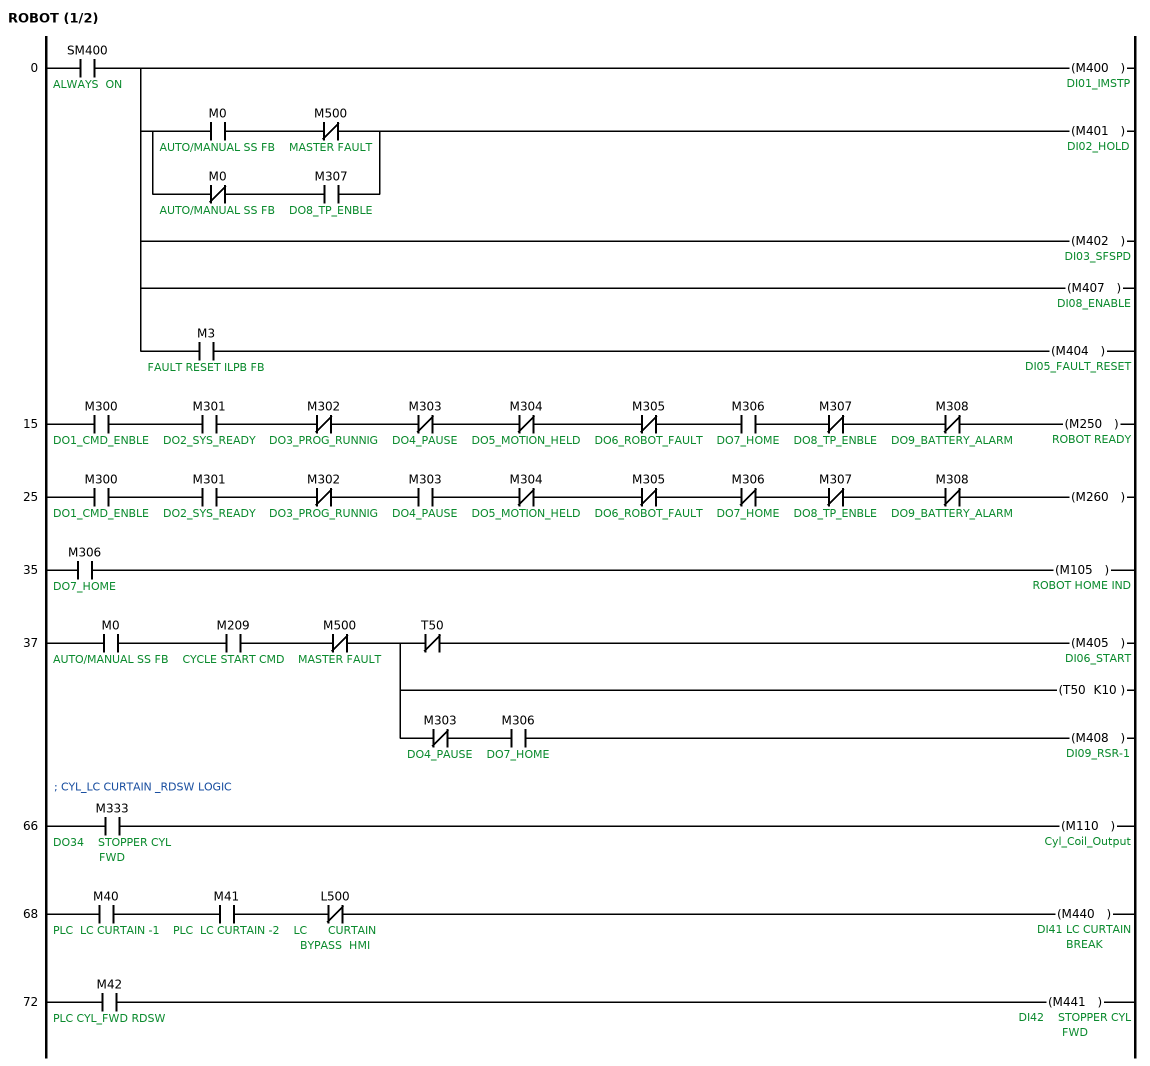
0     LD      SM400  ; ALWAYS  ON
      OUT     M400  ; DI01_IMSTP
      MPS
      LD      M0  ; AUTO/MANUAL SS FB
      ANI     M500  ; MASTER FAULT
      LDI     M0  ; AUTO/MANUAL SS FB
      AND     M307  ; DO8_TP_ENBLE
      ORB
      ANB
      OUT     M401  ; DI02_HOLD
      MPP
      OUT     M402  ; DI03_SFSPD
      OUT     M407  ; DI08_ENABLE
      AND     M3  ; FAULT RESET ILPB FB
      OUT     M404  ; DI05_FAULT_RESET
15    LD      M300  ; DO1_CMD_ENBLE
      AND     M301  ; DO2_SYS_READY
      ANI     M302  ; DO3_PROG_RUNNIG
      ANI     M303  ; DO4_PAUSE
      ANI     M304  ; DO5_MOTION_HELD
      ANI     M305  ; DO6_ROBOT_FAULT
      AND     M306  ; DO7_HOME
      ANI     M307  ; DO8_TP_ENBLE
      ANI     M308  ; DO9_BATTERY_ALARM
      OUT     M250  ; ROBOT READY
25    LD      M300  ; DO1_CMD_ENBLE
      AND     M301  ; DO2_SYS_READY
      ANI     M302  ; DO3_PROG_RUNNIG
      AND     M303  ; DO4_PAUSE
      ANI     M304  ; DO5_MOTION_HELD
      ANI     M305  ; DO6_ROBOT_FAULT
      ANI     M306  ; DO7_HOME
      ANI     M307  ; DO8_TP_ENBLE
      ANI     M308  ; DO9_BATTERY_ALARM
      OUT     M260
35    LD      M306  ; DO7_HOME
      OUT     M105  ; ROBOT HOME IND
37    LD      M0  ; AUTO/MANUAL SS FB
      AND     M209  ; CYCLE START CMD
      ANI     M500  ; MASTER FAULT
      MPS
      ANI     T50
      OUT     M405  ; DI06_START
      MPP
      OUT     T50 K10
      ANI     M303  ; DO4_PAUSE
      AND     M306  ; DO7_HOME
      OUT     M408  ; DI09_RSR-1
; CYL_LC CURTAIN _RDSW LOGIC
66    LD      M333  ; DO34    STOPPER CYL FWD
      OUT     M110  ; Cyl_Coil_Output
68    LD      M40  ; PLC  LC CURTAIN -1
      AND     M41  ; PLC  LC CURTAIN -2
      ANI     L500  ; LC      CURTAIN BYPASS  HMI
      OUT     M440  ; DI41 LC CURTAIN BREAK
72    LD      M42  ; PLC CYL_FWD RDSW
      OUT     M441  ; DI42    STOPPER CYL FWD
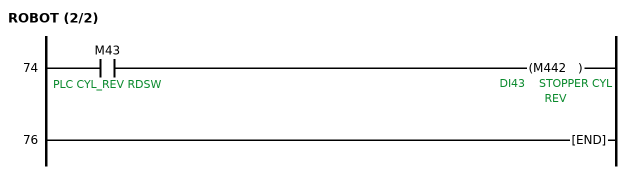
74    LD      M43  ; PLC CYL_REV RDSW
      OUT     M442  ; DI43    STOPPER CYL REV
76    END
END_PROGRAM

PROGRAM CONTROL
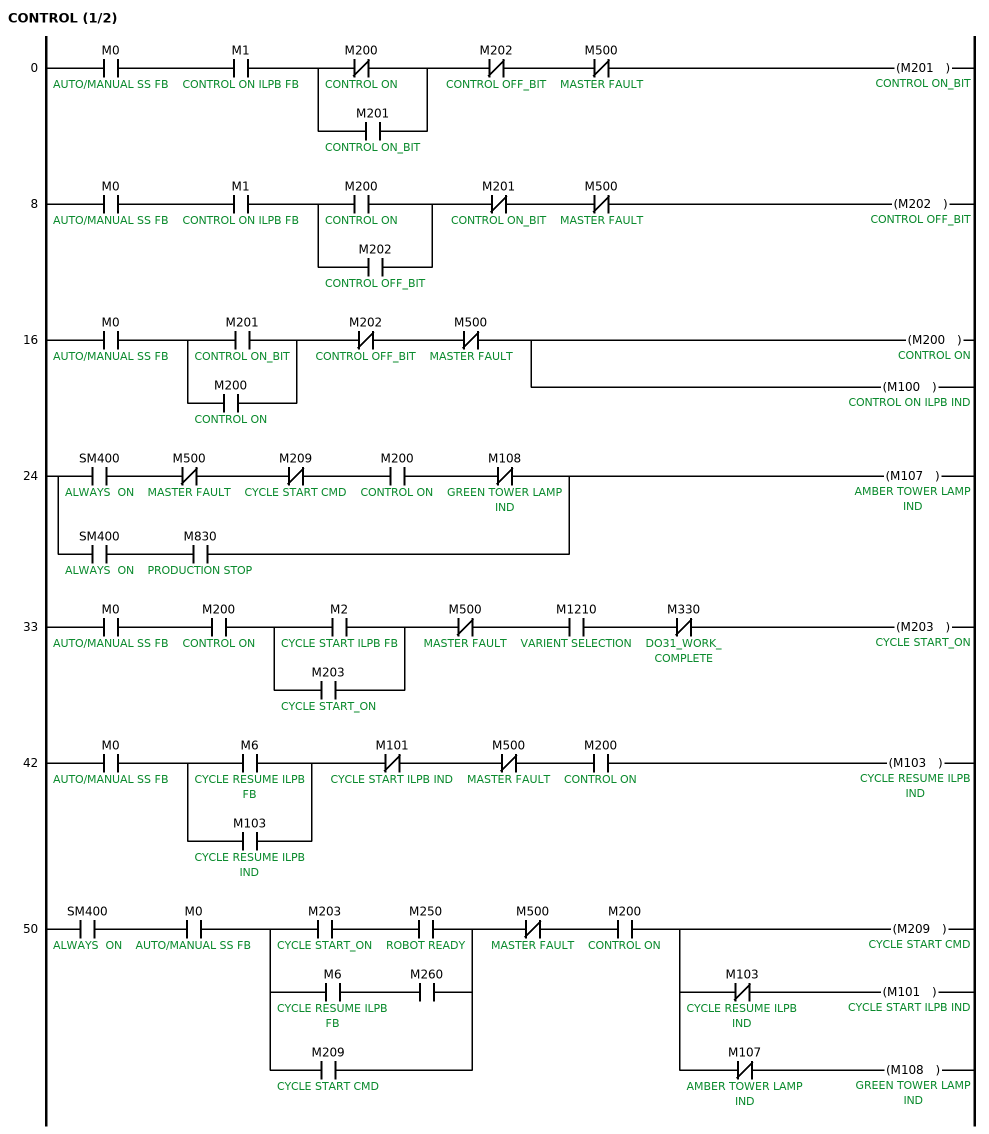
0     LD      M0  ; AUTO/MANUAL SS FB
      AND     M1  ; CONTROL ON ILPB FB
      LDI     M200  ; CONTROL ON
      OR      M201  ; CONTROL ON_BIT
      ANB
      ANI     M202  ; CONTROL OFF_BIT
      ANI     M500  ; MASTER FAULT
      OUT     M201  ; CONTROL ON_BIT
8     LD      M0  ; AUTO/MANUAL SS FB
      AND     M1  ; CONTROL ON ILPB FB
      LD      M200  ; CONTROL ON
      OR      M202  ; CONTROL OFF_BIT
      ANB
      ANI     M201  ; CONTROL ON_BIT
      ANI     M500  ; MASTER FAULT
      OUT     M202  ; CONTROL OFF_BIT
16    LD      M0  ; AUTO/MANUAL SS FB
      LD      M201  ; CONTROL ON_BIT
      OR      M200  ; CONTROL ON
      ANB
      ANI     M202  ; CONTROL OFF_BIT
      ANI     M500  ; MASTER FAULT
      OUT     M200  ; CONTROL ON
      OUT     M100  ; CONTROL ON ILPB IND
24    LD      SM400  ; ALWAYS  ON
      ANI     M500  ; MASTER FAULT
      ANI     M209  ; CYCLE START CMD
      AND     M200  ; CONTROL ON
      ANI     M108  ; GREEN TOWER LAMP IND
      LD      SM400  ; ALWAYS  ON
      AND     M830  ; PRODUCTION STOP
      ORB
      OUT     M107  ; AMBER TOWER LAMP IND
33    LD      M0  ; AUTO/MANUAL SS FB
      AND     M200  ; CONTROL ON
      LD      M2  ; CYCLE START ILPB FB
      OR      M203  ; CYCLE START_ON
      ANB
      ANI     M500  ; MASTER FAULT
      AND     M1210  ; VARIENT SELECTION
      ANI     M330  ; DO31_WORK_COMPLETE
      OUT     M203  ; CYCLE START_ON
42    LD      M0  ; AUTO/MANUAL SS FB
      LD      M6  ; CYCLE RESUME ILPB FB
      OR      M103  ; CYCLE RESUME ILPB IND
      ANB
      ANI     M101  ; CYCLE START ILPB IND
      ANI     M500  ; MASTER FAULT
      AND     M200  ; CONTROL ON
      OUT     M103  ; CYCLE RESUME ILPB IND
50    LD      SM400  ; ALWAYS  ON
      AND     M0  ; AUTO/MANUAL SS FB
      LD      M203  ; CYCLE START_ON
      AND     M250  ; ROBOT READY
      LD      M6  ; CYCLE RESUME ILPB FB
      AND     M260
      ORB
      OR      M209  ; CYCLE START CMD
      ANB
      ANI     M500  ; MASTER FAULT
      AND     M200  ; CONTROL ON
      OUT     M209  ; CYCLE START CMD
      MPS
      ANI     M103  ; CYCLE RESUME ILPB IND
      OUT     M101  ; CYCLE START ILPB IND
      MPP
      ANI     M107  ; AMBER TOWER LAMP IND
      OUT     M108  ; GREEN TOWER LAMP IND
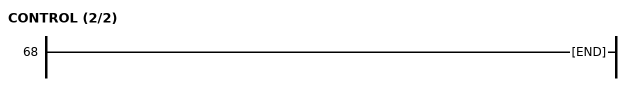
68    END
END_PROGRAM

PROGRAM FAULT
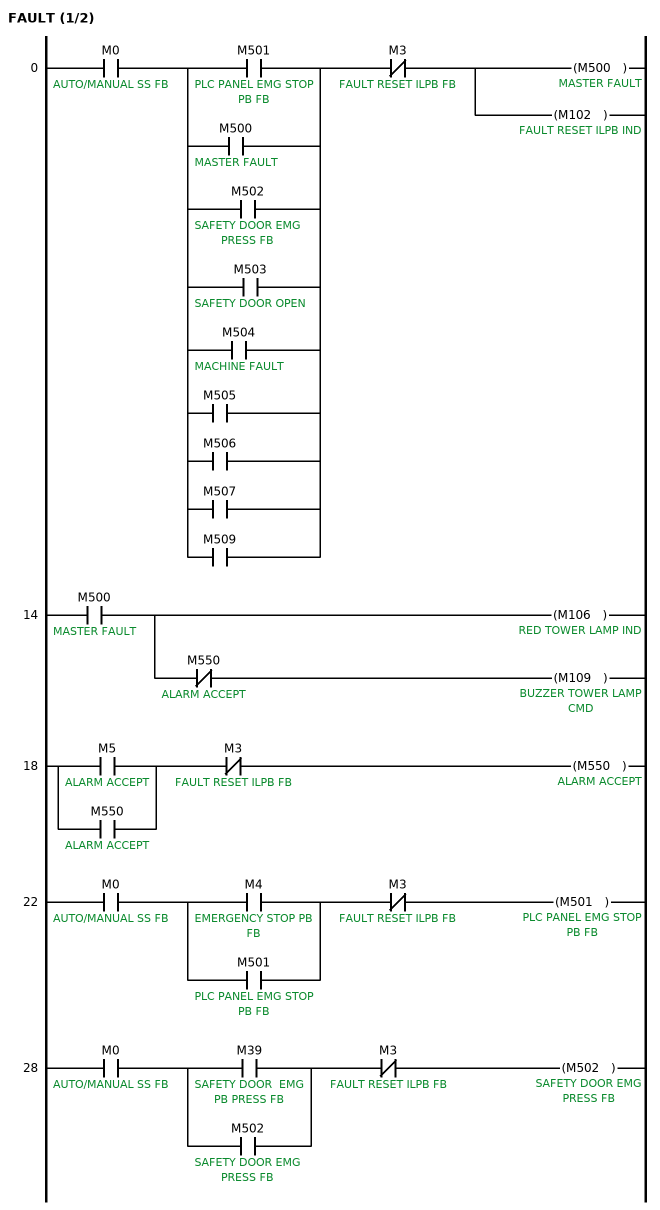
0     LD      M0  ; AUTO/MANUAL SS FB
      LD      M501  ; PLC PANEL EMG STOP PB FB
      OR      M500  ; MASTER FAULT
      OR      M502  ; SAFETY DOOR EMG PRESS FB
      OR      M503  ; SAFETY DOOR OPEN
      OR      M504  ; MACHINE FAULT
      OR      M505
      OR      M506
      OR      M507
      OR      M509
      ANB
      ANI     M3  ; FAULT RESET ILPB FB
      OUT     M500  ; MASTER FAULT
      OUT     M102  ; FAULT RESET ILPB IND
14    LD      M500  ; MASTER FAULT
      OUT     M106  ; RED TOWER LAMP IND
      ANI     M550  ; ALARM ACCEPT
      OUT     M109  ; BUZZER TOWER LAMP CMD
18    LD      M5  ; ALARM ACCEPT
      OR      M550  ; ALARM ACCEPT
      ANI     M3  ; FAULT RESET ILPB FB
      OUT     M550  ; ALARM ACCEPT
22    LD      M0  ; AUTO/MANUAL SS FB
      LD      M4  ; EMERGENCY STOP PB FB
      OR      M501  ; PLC PANEL EMG STOP PB FB
      ANB
      ANI     M3  ; FAULT RESET ILPB FB
      OUT     M501  ; PLC PANEL EMG STOP PB FB
28    LD      M0  ; AUTO/MANUAL SS FB
      LD      M39  ; SAFETY DOOR  EMG PB PRESS FB
      OR      M502  ; SAFETY DOOR EMG PRESS FB
      ANB
      ANI     M3  ; FAULT RESET ILPB FB
      OUT     M502  ; SAFETY DOOR EMG PRESS FB
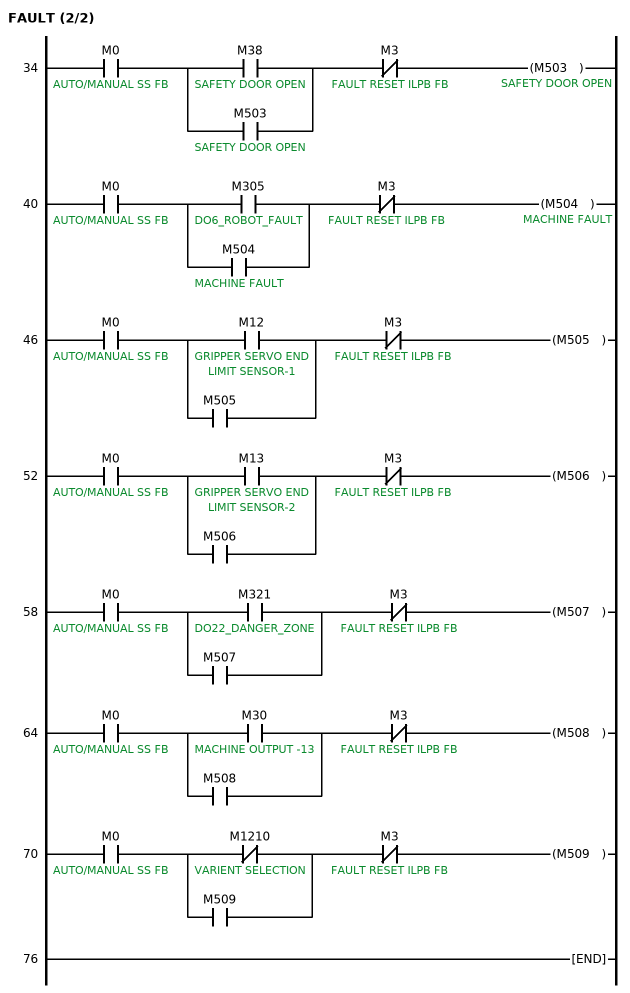
34    LD      M0  ; AUTO/MANUAL SS FB
      LD      M38  ; SAFETY DOOR OPEN
      OR      M503  ; SAFETY DOOR OPEN
      ANB
      ANI     M3  ; FAULT RESET ILPB FB
      OUT     M503  ; SAFETY DOOR OPEN
40    LD      M0  ; AUTO/MANUAL SS FB
      LD      M305  ; DO6_ROBOT_FAULT
      OR      M504  ; MACHINE FAULT
      ANB
      ANI     M3  ; FAULT RESET ILPB FB
      OUT     M504  ; MACHINE FAULT
46    LD      M0  ; AUTO/MANUAL SS FB
      LD      M12  ; GRIPPER SERVO END LIMIT SENSOR-1
      OR      M505
      ANB
      ANI     M3  ; FAULT RESET ILPB FB
      OUT     M505
52    LD      M0  ; AUTO/MANUAL SS FB
      LD      M13  ; GRIPPER SERVO END LIMIT SENSOR-2
      OR      M506
      ANB
      ANI     M3  ; FAULT RESET ILPB FB
      OUT     M506
58    LD      M0  ; AUTO/MANUAL SS FB
      LD      M321  ; DO22_DANGER_ZONE
      OR      M507
      ANB
      ANI     M3  ; FAULT RESET ILPB FB
      OUT     M507
64    LD      M0  ; AUTO/MANUAL SS FB
      LD      M30  ; MACHINE OUTPUT -13
      OR      M508
      ANB
      ANI     M3  ; FAULT RESET ILPB FB
      OUT     M508
70    LD      M0  ; AUTO/MANUAL SS FB
      LDI     M1210  ; VARIENT SELECTION
      OR      M509
      ANB
      ANI     M3  ; FAULT RESET ILPB FB
      OUT     M509
76    END
END_PROGRAM

PROGRAM MACHINE
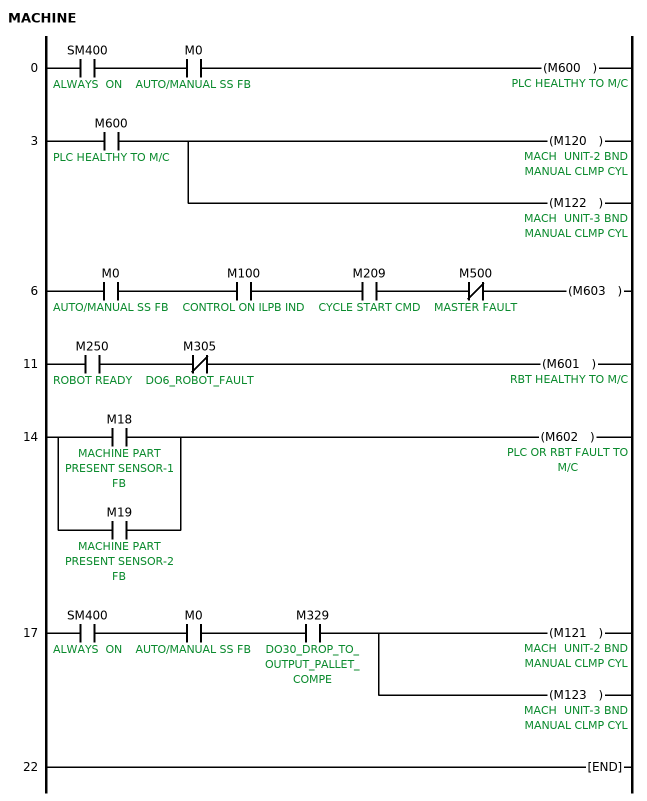
0     LD      SM400  ; ALWAYS  ON
      AND     M0  ; AUTO/MANUAL SS FB
      OUT     M600  ; PLC HEALTHY TO M/C
3     LD      M600  ; PLC HEALTHY TO M/C
      OUT     M120  ; MACH  UNIT-2 BND MANUAL CLMP CYL
      OUT     M122  ; MACH  UNIT-3 BND MANUAL CLMP CYL
6     LD      M0  ; AUTO/MANUAL SS FB
      AND     M100  ; CONTROL ON ILPB IND
      AND     M209  ; CYCLE START CMD
      ANI     M500  ; MASTER FAULT
      OUT     M603
11    LD      M250  ; ROBOT READY
      ANI     M305  ; DO6_ROBOT_FAULT
      OUT     M601  ; RBT HEALTHY TO M/C
14    LD      M18  ; MACHINE PART PRESENT SENSOR-1 FB
      OR      M19  ; MACHINE PART PRESENT SENSOR-2 FB
      OUT     M602  ; PLC OR RBT FAULT TO M/C
17    LD      SM400  ; ALWAYS  ON
      AND     M0  ; AUTO/MANUAL SS FB
      AND     M329  ; DO30_DROP_TO_OUTPUT_PALLET_COMPE
      OUT     M121  ; MACH  UNIT-2 BND MANUAL CLMP CYL
      OUT     M123  ; MACH  UNIT-3 BND MANUAL CLMP CYL
22    END
END_PROGRAM

PROGRAM HMI
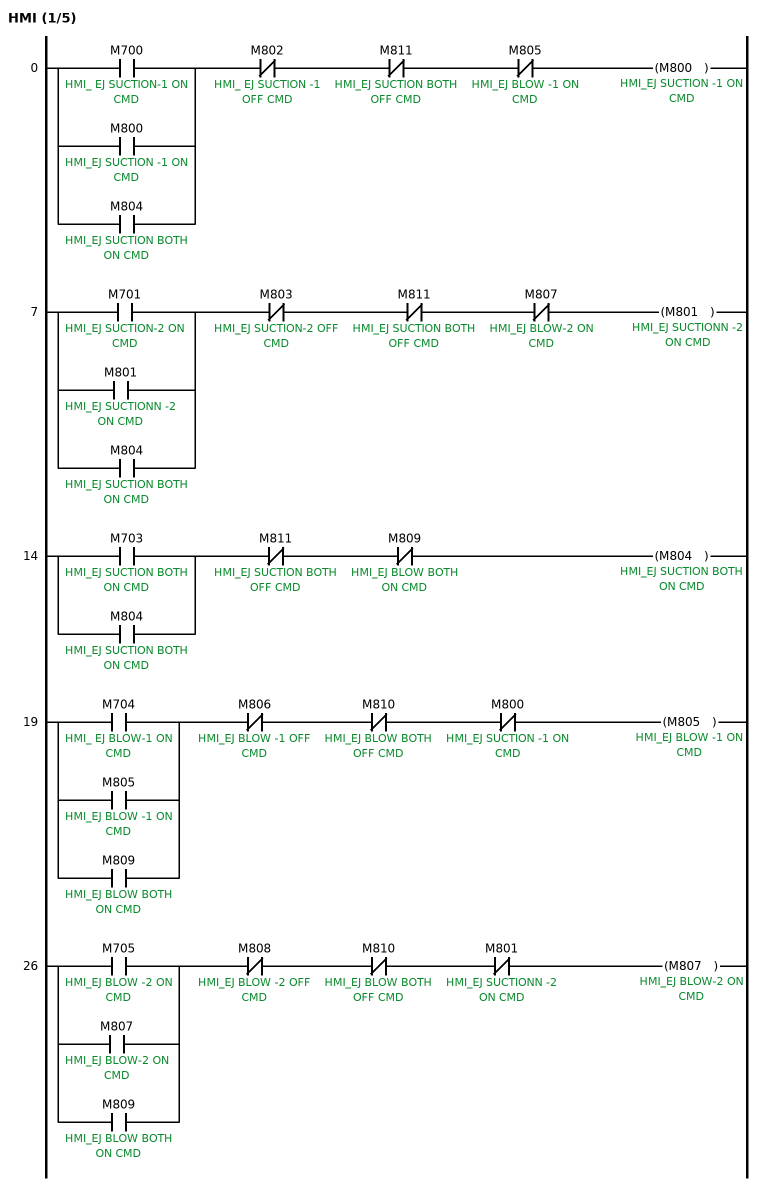
0     LD      M700  ; HMI_ EJ SUCTION-1 ON CMD
      OR      M800  ; HMI_EJ SUCTION -1 ON CMD
      OR      M804  ; HMI_EJ SUCTION BOTH ON CMD
      ANI     M802  ; HMI_ EJ SUCTION -1 OFF CMD
      ANI     M811  ; HMI_EJ SUCTION BOTH OFF CMD
      ANI     M805  ; HMI_EJ BLOW -1 ON CMD
      OUT     M800  ; HMI_EJ SUCTION -1 ON CMD
7     LD      M701  ; HMI_EJ SUCTION-2 ON CMD
      OR      M801  ; HMI_EJ SUCTIONN -2 ON CMD
      OR      M804  ; HMI_EJ SUCTION BOTH ON CMD
      ANI     M803  ; HMI_EJ SUCTION-2 OFF CMD
      ANI     M811  ; HMI_EJ SUCTION BOTH OFF CMD
      ANI     M807  ; HMI_EJ BLOW-2 ON CMD
      OUT     M801  ; HMI_EJ SUCTIONN -2 ON CMD
14    LD      M703  ; HMI_EJ SUCTION BOTH ON CMD
      OR      M804  ; HMI_EJ SUCTION BOTH ON CMD
      ANI     M811  ; HMI_EJ SUCTION BOTH OFF CMD
      ANI     M809  ; HMI_EJ BLOW BOTH ON CMD
      OUT     M804  ; HMI_EJ SUCTION BOTH ON CMD
19    LD      M704  ; HMI_ EJ BLOW-1 ON CMD
      OR      M805  ; HMI_EJ BLOW -1 ON CMD
      OR      M809  ; HMI_EJ BLOW BOTH ON CMD
      ANI     M806  ; HMI_EJ BLOW -1 OFF CMD
      ANI     M810  ; HMI_EJ BLOW BOTH OFF CMD
      ANI     M800  ; HMI_EJ SUCTION -1 ON CMD
      OUT     M805  ; HMI_EJ BLOW -1 ON CMD
26    LD      M705  ; HMI_EJ BLOW -2 ON CMD
      OR      M807  ; HMI_EJ BLOW-2 ON CMD
      OR      M809  ; HMI_EJ BLOW BOTH ON CMD
      ANI     M808  ; HMI_EJ BLOW -2 OFF CMD
      ANI     M810  ; HMI_EJ BLOW BOTH OFF CMD
      ANI     M801  ; HMI_EJ SUCTIONN -2 ON CMD
      OUT     M807  ; HMI_EJ BLOW-2 ON CMD
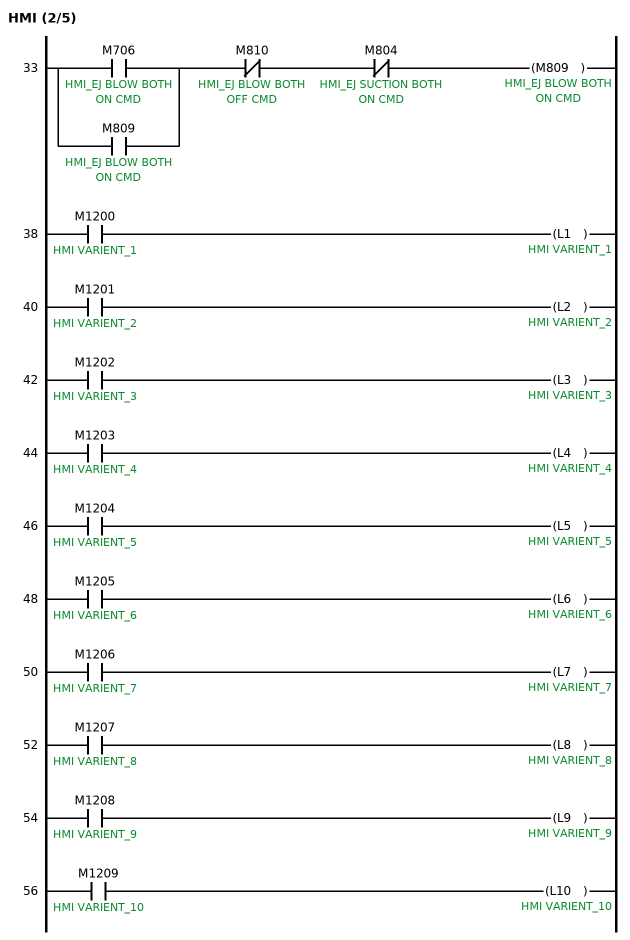
33    LD      M706  ; HMI_EJ BLOW BOTH ON CMD
      OR      M809  ; HMI_EJ BLOW BOTH ON CMD
      ANI     M810  ; HMI_EJ BLOW BOTH OFF CMD
      ANI     M804  ; HMI_EJ SUCTION BOTH ON CMD
      OUT     M809  ; HMI_EJ BLOW BOTH ON CMD
38    LD      M1200  ; HMI VARIENT_1
      OUT     L1  ; HMI VARIENT_1
40    LD      M1201  ; HMI VARIENT_2
      OUT     L2  ; HMI VARIENT_2
42    LD      M1202  ; HMI VARIENT_3
      OUT     L3  ; HMI VARIENT_3
44    LD      M1203  ; HMI VARIENT_4
      OUT     L4  ; HMI VARIENT_4
46    LD      M1204  ; HMI VARIENT_5
      OUT     L5  ; HMI VARIENT_5
48    LD      M1205  ; HMI VARIENT_6
      OUT     L6  ; HMI VARIENT_6
50    LD      M1206  ; HMI VARIENT_7
      OUT     L7  ; HMI VARIENT_7
52    LD      M1207  ; HMI VARIENT_8
      OUT     L8  ; HMI VARIENT_8
54    LD      M1208  ; HMI VARIENT_9
      OUT     L9  ; HMI VARIENT_9
56    LD      M1209  ; HMI VARIENT_10
      OUT     L10  ; HMI VARIENT_10
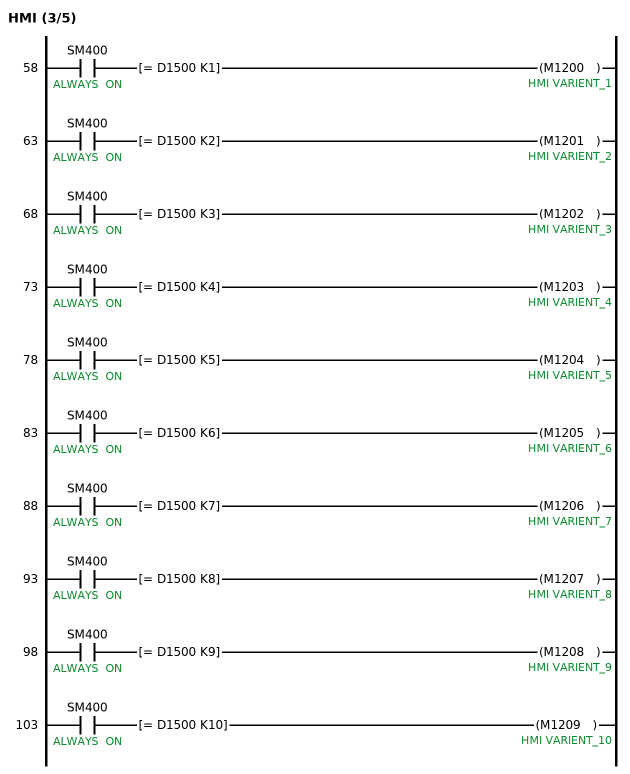
58    LD      SM400  ; ALWAYS  ON
      AND=    D1500 K1
      OUT     M1200  ; HMI VARIENT_1
63    LD      SM400  ; ALWAYS  ON
      AND=    D1500 K2
      OUT     M1201  ; HMI VARIENT_2
68    LD      SM400  ; ALWAYS  ON
      AND=    D1500 K3
      OUT     M1202  ; HMI VARIENT_3
73    LD      SM400  ; ALWAYS  ON
      AND=    D1500 K4
      OUT     M1203  ; HMI VARIENT_4
78    LD      SM400  ; ALWAYS  ON
      AND=    D1500 K5
      OUT     M1204  ; HMI VARIENT_5
83    LD      SM400  ; ALWAYS  ON
      AND=    D1500 K6
      OUT     M1205  ; HMI VARIENT_6
88    LD      SM400  ; ALWAYS  ON
      AND=    D1500 K7
      OUT     M1206  ; HMI VARIENT_7
93    LD      SM400  ; ALWAYS  ON
      AND=    D1500 K8
      OUT     M1207  ; HMI VARIENT_8
98    LD      SM400  ; ALWAYS  ON
      AND=    D1500 K9
      OUT     M1208  ; HMI VARIENT_9
103   LD      SM400  ; ALWAYS  ON
      AND=    D1500 K10
      OUT     M1209  ; HMI VARIENT_10
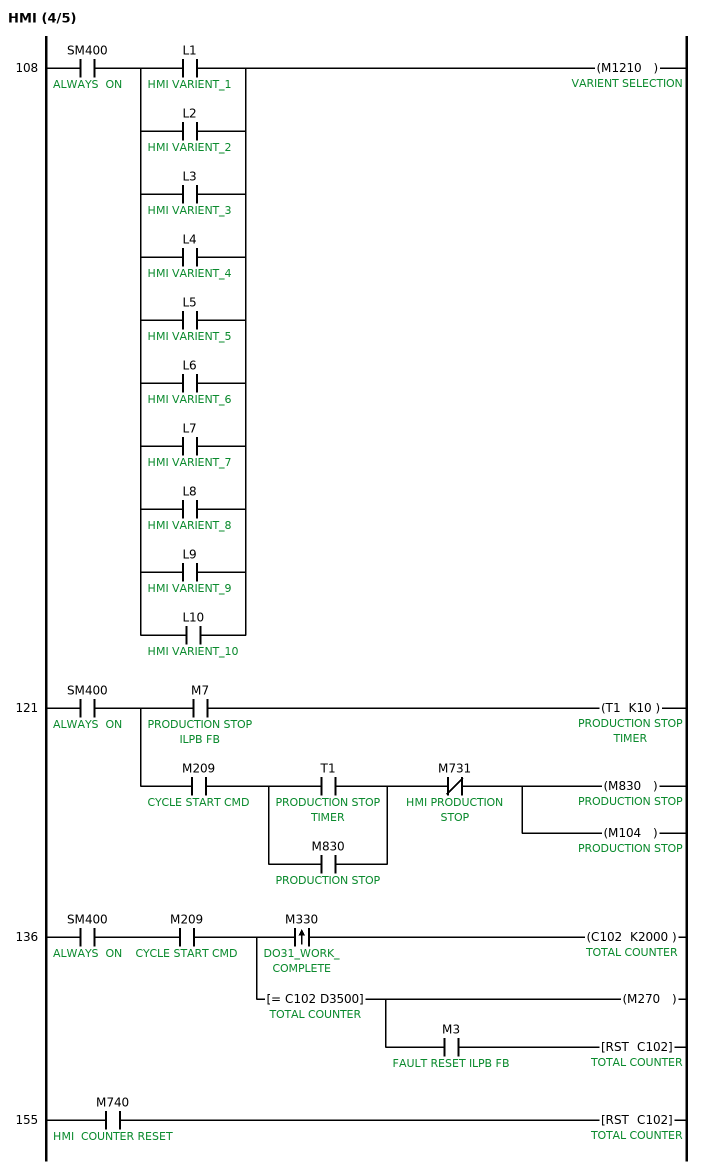
108   LD      SM400  ; ALWAYS  ON
      LD      L1  ; HMI VARIENT_1
      OR      L2  ; HMI VARIENT_2
      OR      L3  ; HMI VARIENT_3
      OR      L4  ; HMI VARIENT_4
      OR      L5  ; HMI VARIENT_5
      OR      L6  ; HMI VARIENT_6
      OR      L7  ; HMI VARIENT_7
      OR      L8  ; HMI VARIENT_8
      OR      L9  ; HMI VARIENT_9
      OR      L10  ; HMI VARIENT_10
      ANB
      OUT     M1210  ; VARIENT SELECTION
121   LD      SM400  ; ALWAYS  ON
      MPS
      AND     M7  ; PRODUCTION STOP ILPB FB
      OUT     T1 K10  ; PRODUCTION STOP TIMER
      MPP
      AND     M209  ; CYCLE START CMD
      LD      T1  ; PRODUCTION STOP TIMER
      OR      M830  ; PRODUCTION STOP
      ANB
      ANI     M731  ; HMI PRODUCTION STOP
      OUT     M830  ; PRODUCTION STOP
      OUT     M104  ; PRODUCTION STOP
136   LD      SM400  ; ALWAYS  ON
      AND     M209  ; CYCLE START CMD
      MPS
      ANDP    M330  ; DO31_WORK_COMPLETE
      OUT     C102 K2000  ; TOTAL COUNTER
      MPP
      AND=    C102 D3500  ; TOTAL COUNTER
      OUT     M270
      AND     M3  ; FAULT RESET ILPB FB
      RST     C102  ; TOTAL COUNTER
155   LD      M740  ; HMI  COUNTER RESET
      RST     C102  ; TOTAL COUNTER
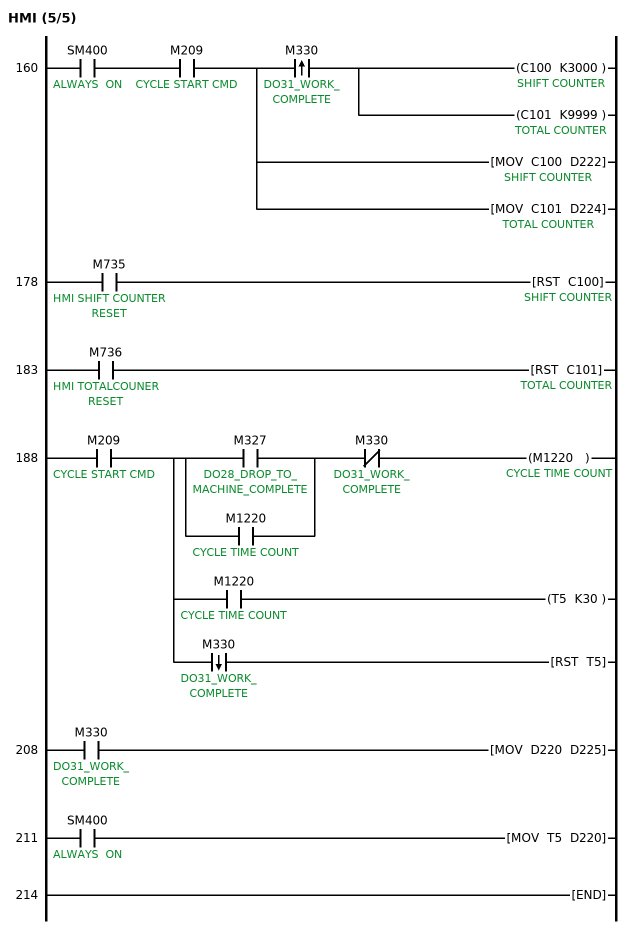
160   LD      SM400  ; ALWAYS  ON
      AND     M209  ; CYCLE START CMD
      MPS
      ANDP    M330  ; DO31_WORK_COMPLETE
      OUT     C100 K3000  ; SHIFT COUNTER
      OUT     C101 K9999  ; TOTAL COUNTER
      MPP
      MOV     C100 D222
      MOV     C101 D224
178   LD      M735  ; HMI SHIFT COUNTER RESET
      RST     C100  ; SHIFT COUNTER
183   LD      M736  ; HMI TOTALCOUNER RESET
      RST     C101  ; TOTAL COUNTER
188   LD      M209  ; CYCLE START CMD
      MPS
      LD      M327  ; DO28_DROP_TO_MACHINE_COMPLETE
      OR      M1220  ; CYCLE TIME COUNT
      ANB
      ANI     M330  ; DO31_WORK_COMPLETE
      OUT     M1220  ; CYCLE TIME COUNT
      MRD
      AND     M1220  ; CYCLE TIME COUNT
      OUT     T5 K30
      MPP
      ANDF    M330  ; DO31_WORK_COMPLETE
      RST     T5
208   LD      M330  ; DO31_WORK_COMPLETE
      MOV     D220 D225
211   LD      SM400  ; ALWAYS  ON
      MOV     T5 D220
214   END
END_PROGRAM

PROGRAM RBT_INP
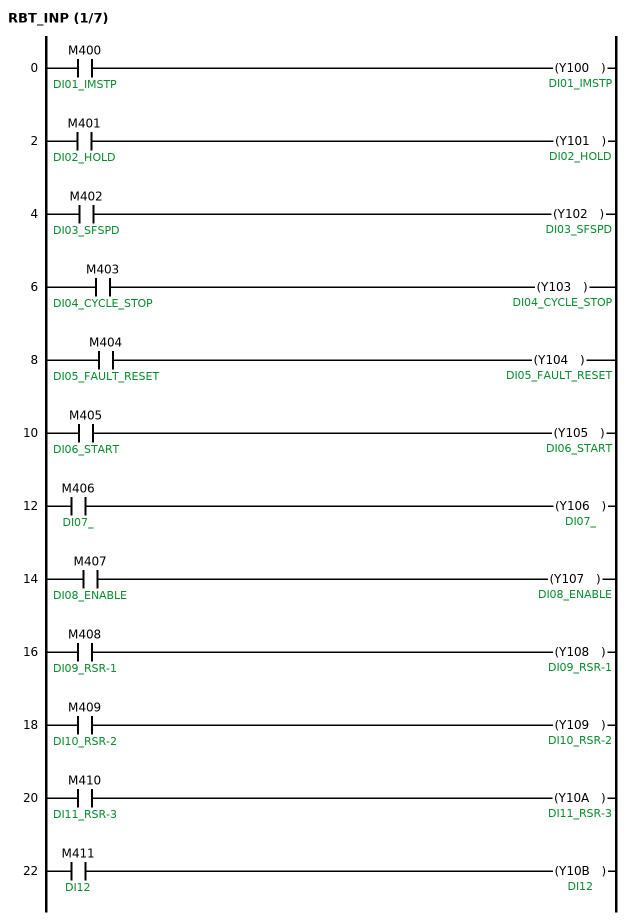
0     LD      M400  ; DI01_IMSTP
      OUT     Y100  ; DI01_IMSTP
2     LD      M401  ; DI02_HOLD
      OUT     Y101  ; DI02_HOLD
4     LD      M402  ; DI03_SFSPD
      OUT     Y102  ; DI03_SFSPD
6     LD      M403  ; DI04_CYCLE_STOP
      OUT     Y103  ; DI04_CYCLE_STOP
8     LD      M404  ; DI05_FAULT_RESET
      OUT     Y104  ; DI05_FAULT_RESET
10    LD      M405  ; DI06_START
      OUT     Y105  ; DI06_START
12    LD      M406  ; DI07_
      OUT     Y106  ; DI07_
14    LD      M407  ; DI08_ENABLE
      OUT     Y107  ; DI08_ENABLE
16    LD      M408  ; DI09_RSR-1
      OUT     Y108  ; DI09_RSR-1
18    LD      M409  ; DI10_RSR-2
      OUT     Y109  ; DI10_RSR-2
20    LD      M410  ; DI11_RSR-3
      OUT     Y10A  ; DI11_RSR-3
22    LD      M411  ; DI12
      OUT     Y10B  ; DI12
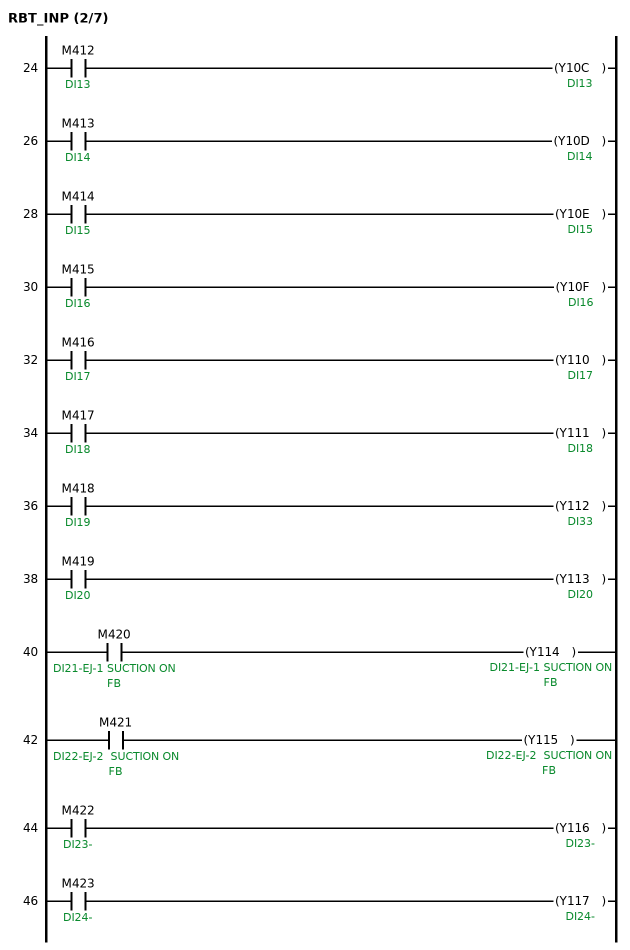
24    LD      M412  ; DI13
      OUT     Y10C  ; DI13
26    LD      M413  ; DI14
      OUT     Y10D  ; DI14
28    LD      M414  ; DI15
      OUT     Y10E  ; DI15
30    LD      M415  ; DI16
      OUT     Y10F  ; DI16
32    LD      M416  ; DI17
      OUT     Y110  ; DI17
34    LD      M417  ; DI18
      OUT     Y111  ; DI18
36    LD      M418  ; DI19
      OUT     Y112  ; DI33
38    LD      M419  ; DI20
      OUT     Y113  ; DI20
40    LD      M420  ; DI21-EJ-1 SUCTION ON FB
      OUT     Y114  ; DI21-EJ-1 SUCTION ON FB
42    LD      M421  ; DI22-EJ-2  SUCTION ON FB
      OUT     Y115  ; DI22-EJ-2  SUCTION ON FB
44    LD      M422  ; DI23-
      OUT     Y116  ; DI23-
46    LD      M423  ; DI24-
      OUT     Y117  ; DI24-
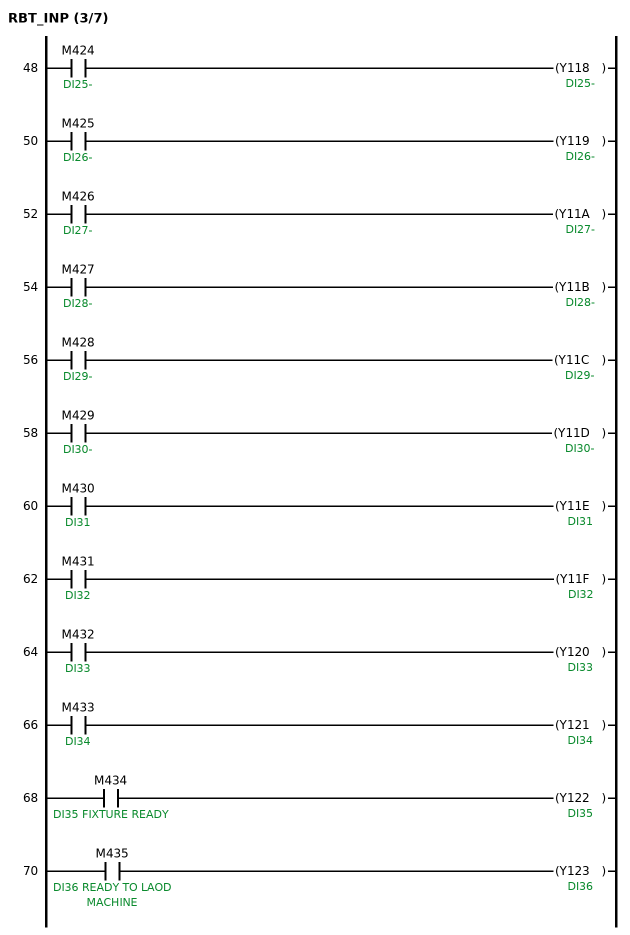
48    LD      M424  ; DI25-
      OUT     Y118  ; DI25-
50    LD      M425  ; DI26-
      OUT     Y119  ; DI26-
52    LD      M426  ; DI27-
      OUT     Y11A  ; DI27-
54    LD      M427  ; DI28-
      OUT     Y11B  ; DI28-
56    LD      M428  ; DI29-
      OUT     Y11C  ; DI29-
58    LD      M429  ; DI30-
      OUT     Y11D  ; DI30-
60    LD      M430  ; DI31
      OUT     Y11E  ; DI31
62    LD      M431  ; DI32
      OUT     Y11F  ; DI32
64    LD      M432  ; DI33
      OUT     Y120  ; DI33
66    LD      M433  ; DI34
      OUT     Y121  ; DI34
68    LD      M434  ; DI35 FIXTURE READY
      OUT     Y122  ; DI35
70    LD      M435  ; DI36 READY TO LAOD MACHINE
      OUT     Y123  ; DI36
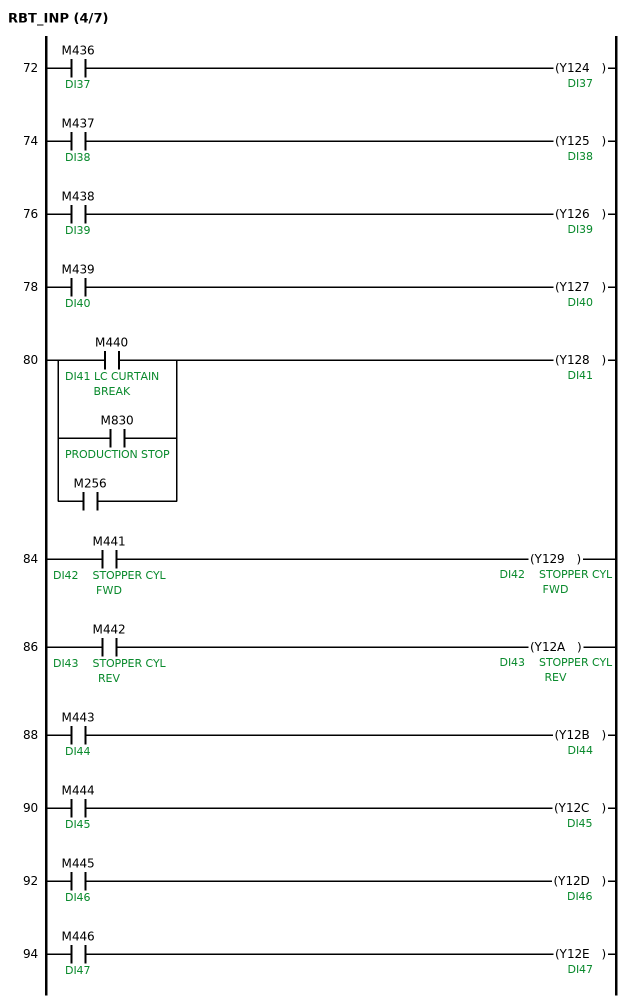
72    LD      M436  ; DI37
      OUT     Y124  ; DI37
74    LD      M437  ; DI38
      OUT     Y125  ; DI38
76    LD      M438  ; DI39
      OUT     Y126  ; DI39
78    LD      M439  ; DI40
      OUT     Y127  ; DI40
80    LD      M440  ; DI41 LC CURTAIN BREAK
      OR      M830  ; PRODUCTION STOP
      OR      M256
      OUT     Y128  ; DI41
84    LD      M441  ; DI42    STOPPER CYL FWD
      OUT     Y129  ; DI42    STOPPER CYL FWD
86    LD      M442  ; DI43    STOPPER CYL REV
      OUT     Y12A  ; DI43    STOPPER CYL REV
88    LD      M443  ; DI44
      OUT     Y12B  ; DI44
90    LD      M444  ; DI45
      OUT     Y12C  ; DI45
92    LD      M445  ; DI46
      OUT     Y12D  ; DI46
94    LD      M446  ; DI47
      OUT     Y12E  ; DI47
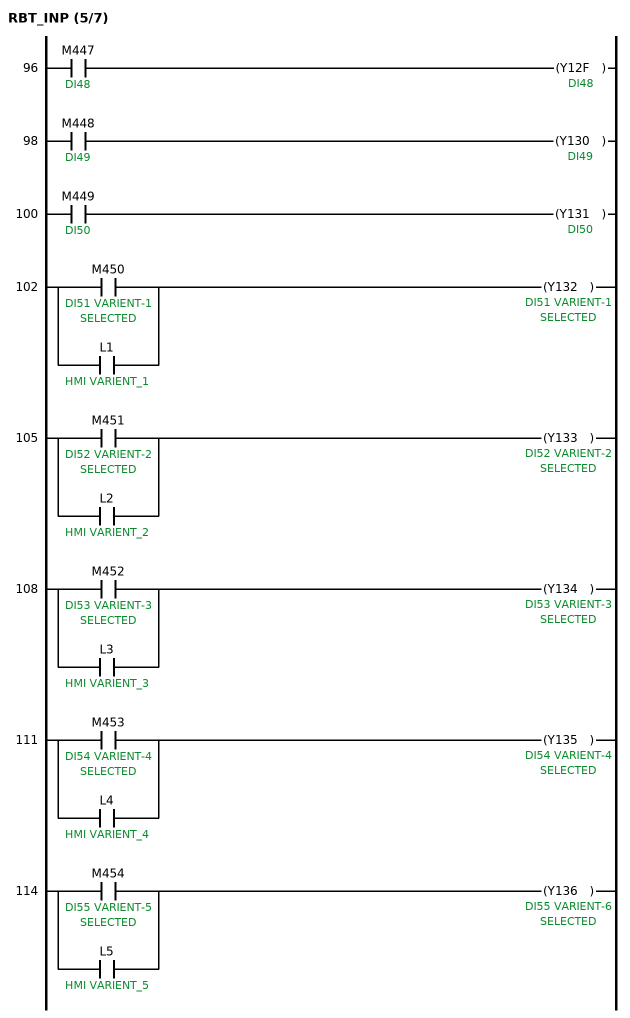
96    LD      M447  ; DI48
      OUT     Y12F  ; DI48
98    LD      M448  ; DI49
      OUT     Y130  ; DI49
100   LD      M449  ; DI50
      OUT     Y131  ; DI50
102   LD      M450  ; DI51 VARIENT-1 SELECTED
      OR      L1  ; HMI VARIENT_1
      OUT     Y132  ; DI51 VARIENT-1 SELECTED
105   LD      M451  ; DI52 VARIENT-2 SELECTED
      OR      L2  ; HMI VARIENT_2
      OUT     Y133  ; DI52 VARIENT-2 SELECTED
108   LD      M452  ; DI53 VARIENT-3 SELECTED
      OR      L3  ; HMI VARIENT_3
      OUT     Y134  ; DI53 VARIENT-3 SELECTED
111   LD      M453  ; DI54 VARIENT-4 SELECTED
      OR      L4  ; HMI VARIENT_4
      OUT     Y135  ; DI54 VARIENT-4 SELECTED
114   LD      M454  ; DI55 VARIENT-5 SELECTED
      OR      L5  ; HMI VARIENT_5
      OUT     Y136  ; DI55 VARIENT-6 SELECTED
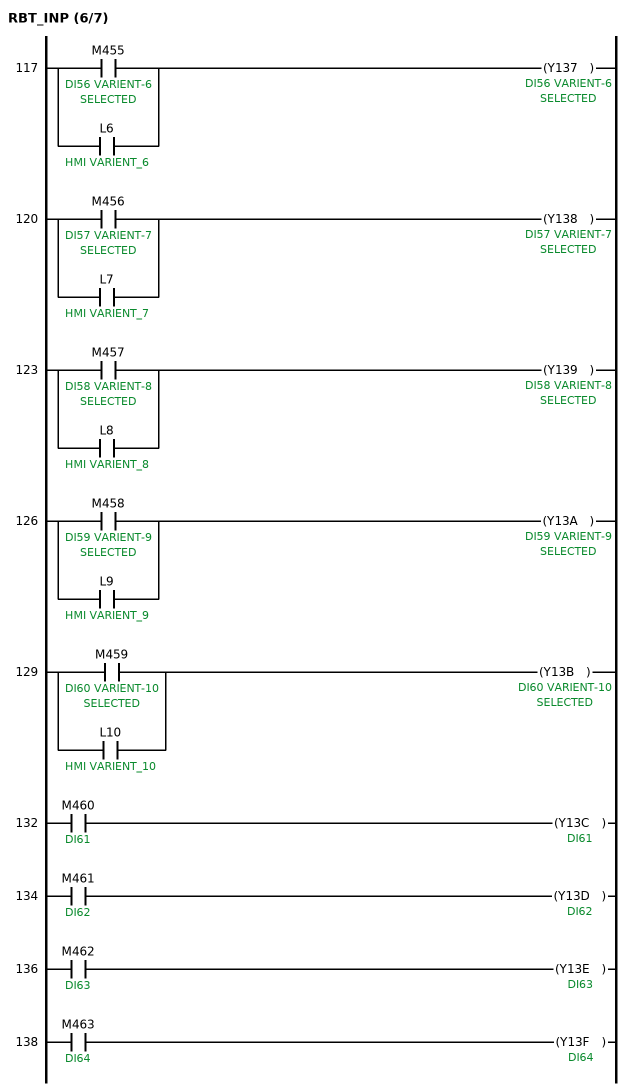
117   LD      M455  ; DI56 VARIENT-6 SELECTED
      OR      L6  ; HMI VARIENT_6
      OUT     Y137  ; DI56 VARIENT-6 SELECTED
120   LD      M456  ; DI57 VARIENT-7 SELECTED
      OR      L7  ; HMI VARIENT_7
      OUT     Y138  ; DI57 VARIENT-7 SELECTED
123   LD      M457  ; DI58 VARIENT-8 SELECTED
      OR      L8  ; HMI VARIENT_8
      OUT     Y139  ; DI58 VARIENT-8 SELECTED
126   LD      M458  ; DI59 VARIENT-9 SELECTED
      OR      L9  ; HMI VARIENT_9
      OUT     Y13A  ; DI59 VARIENT-9 SELECTED
129   LD      M459  ; DI60 VARIENT-10 SELECTED
      OR      L10  ; HMI VARIENT_10
      OUT     Y13B  ; DI60 VARIENT-10 SELECTED
132   LD      M460  ; DI61
      OUT     Y13C  ; DI61
134   LD      M461  ; DI62
      OUT     Y13D  ; DI62
136   LD      M462  ; DI63
      OUT     Y13E  ; DI63
138   LD      M463  ; DI64
      OUT     Y13F  ; DI64
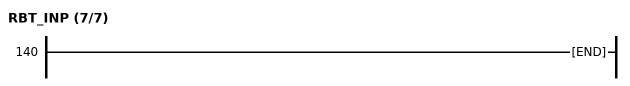
140   END
END_PROGRAM

PROGRAM PLC-INP
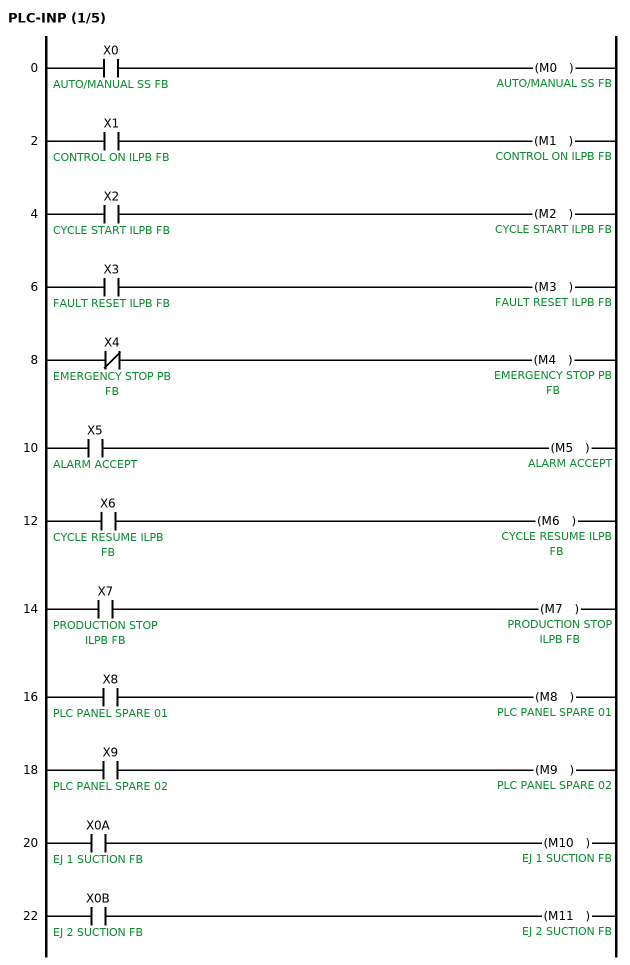
0     LD      X0  ; AUTO/MANUAL SS FB
      OUT     M0  ; AUTO/MANUAL SS FB
2     LD      X1  ; CONTROL ON ILPB FB
      OUT     M1  ; CONTROL ON ILPB FB
4     LD      X2  ; CYCLE START ILPB FB
      OUT     M2  ; CYCLE START ILPB FB
6     LD      X3  ; FAULT RESET ILPB FB
      OUT     M3  ; FAULT RESET ILPB FB
8     LDI     X4  ; EMERGENCY STOP PB FB
      OUT     M4  ; EMERGENCY STOP PB FB
10    LD      X5  ; ALARM ACCEPT
      OUT     M5  ; ALARM ACCEPT
12    LD      X6  ; CYCLE RESUME ILPB FB
      OUT     M6  ; CYCLE RESUME ILPB FB
14    LD      X7  ; PRODUCTION STOP ILPB FB
      OUT     M7  ; PRODUCTION STOP ILPB FB
16    LD      X8  ; PLC PANEL SPARE 01
      OUT     M8  ; PLC PANEL SPARE 01
18    LD      X9  ; PLC PANEL SPARE 02
      OUT     M9  ; PLC PANEL SPARE 02
20    LD      X0A  ; EJ 1 SUCTION FB
      OUT     M10  ; EJ 1 SUCTION FB
22    LD      X0B  ; EJ 2 SUCTION FB
      OUT     M11  ; EJ 2 SUCTION FB
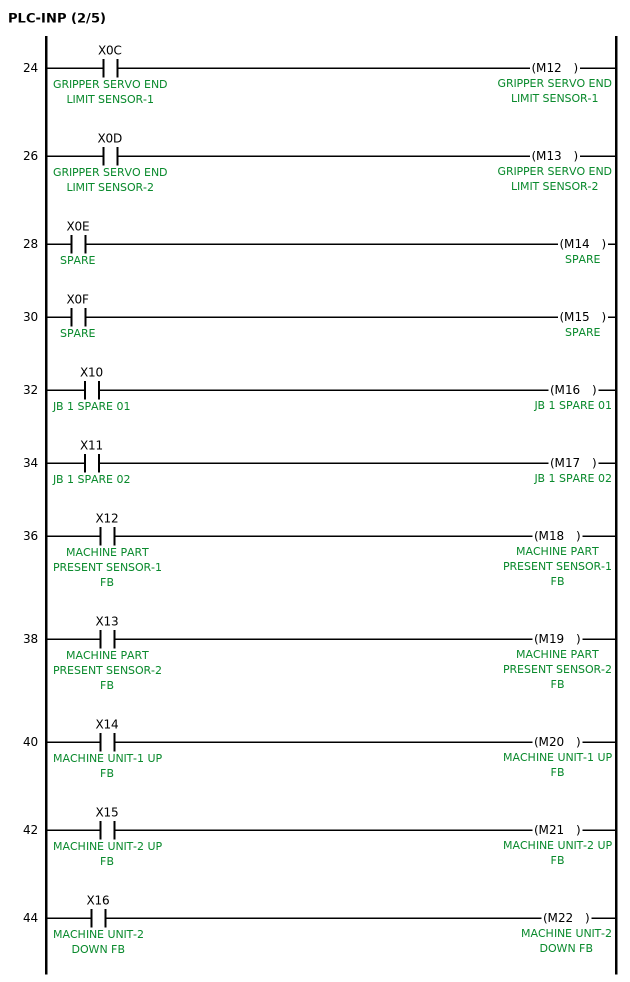
24    LD      X0C  ; GRIPPER SERVO END LIMIT SENSOR-1
      OUT     M12  ; GRIPPER SERVO END LIMIT SENSOR-1
26    LD      X0D  ; GRIPPER SERVO END LIMIT SENSOR-2
      OUT     M13  ; GRIPPER SERVO END LIMIT SENSOR-2
28    LD      X0E  ; SPARE
      OUT     M14  ; SPARE
30    LD      X0F  ; SPARE
      OUT     M15  ; SPARE
32    LD      X10  ; JB 1 SPARE 01
      OUT     M16  ; JB 1 SPARE 01
34    LD      X11  ; JB 1 SPARE 02
      OUT     M17  ; JB 1 SPARE 02
36    LD      X12  ; MACHINE PART PRESENT SENSOR-1 FB
      OUT     M18  ; MACHINE PART PRESENT SENSOR-1 FB
38    LD      X13  ; MACHINE PART PRESENT SENSOR-2 FB
      OUT     M19  ; MACHINE PART PRESENT SENSOR-2 FB
40    LD      X14  ; MACHINE UNIT-1 UP FB
      OUT     M20  ; MACHINE UNIT-1 UP FB
42    LD      X15  ; MACHINE UNIT-2 UP FB
      OUT     M21  ; MACHINE UNIT-2 UP FB
44    LD      X16  ; MACHINE UNIT-2 DOWN FB
      OUT     M22  ; MACHINE UNIT-2 DOWN FB
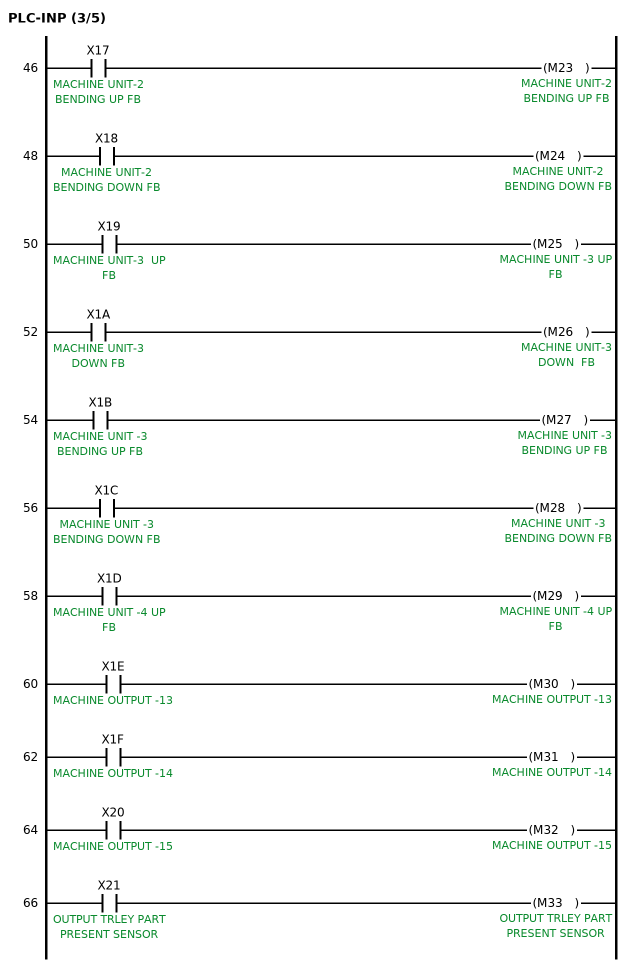
46    LD      X17  ; MACHINE UNIT-2 BENDING UP FB
      OUT     M23  ; MACHINE UNIT-2 BENDING UP FB
48    LD      X18  ; MACHINE UNIT-2 BENDING DOWN FB
      OUT     M24  ; MACHINE UNIT-2 BENDING DOWN FB
50    LD      X19  ; MACHINE UNIT-3  UP FB
      OUT     M25  ; MACHINE UNIT -3 UP FB
52    LD      X1A  ; MACHINE UNIT-3 DOWN FB
      OUT     M26  ; MACHINE UNIT-3 DOWN  FB
54    LD      X1B  ; MACHINE UNIT -3 BENDING UP FB
      OUT     M27  ; MACHINE UNIT -3 BENDING UP FB
56    LD      X1C  ; MACHINE UNIT -3 BENDING DOWN FB
      OUT     M28  ; MACHINE UNIT -3 BENDING DOWN FB
58    LD      X1D  ; MACHINE UNIT -4 UP FB
      OUT     M29  ; MACHINE UNIT -4 UP FB
60    LD      X1E  ; MACHINE OUTPUT -13
      OUT     M30  ; MACHINE OUTPUT -13
62    LD      X1F  ; MACHINE OUTPUT -14
      OUT     M31  ; MACHINE OUTPUT -14
64    LD      X20  ; MACHINE OUTPUT -15
      OUT     M32  ; MACHINE OUTPUT -15
66    LD      X21  ; OUTPUT TRLEY PART PRESENT SENSOR
      OUT     M33  ; OUTPUT TRLEY PART PRESENT SENSOR
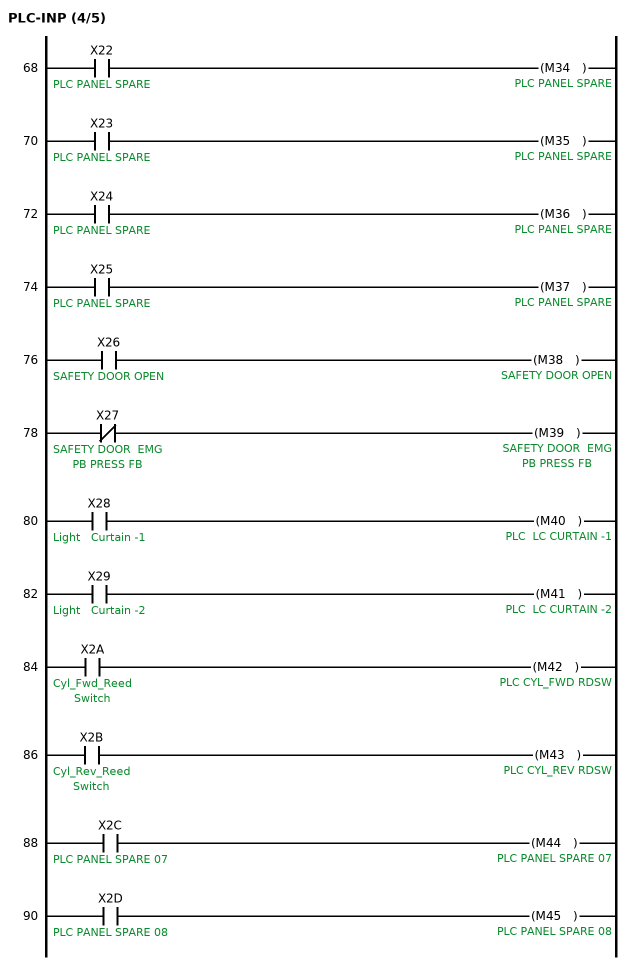
68    LD      X22  ; PLC PANEL SPARE
      OUT     M34  ; PLC PANEL SPARE
70    LD      X23  ; PLC PANEL SPARE
      OUT     M35  ; PLC PANEL SPARE
72    LD      X24  ; PLC PANEL SPARE
      OUT     M36  ; PLC PANEL SPARE
74    LD      X25  ; PLC PANEL SPARE
      OUT     M37  ; PLC PANEL SPARE
76    LD      X26  ; SAFETY DOOR OPEN
      OUT     M38  ; SAFETY DOOR OPEN
78    LDI     X27  ; SAFETY DOOR  EMG PB PRESS FB
      OUT     M39  ; SAFETY DOOR  EMG PB PRESS FB
80    LD      X28  ; Light   Curtain -1
      OUT     M40  ; PLC  LC CURTAIN -1
82    LD      X29  ; Light   Curtain -2
      OUT     M41  ; PLC  LC CURTAIN -2
84    LD      X2A  ; Cyl_Fwd_Reed    Switch
      OUT     M42  ; PLC CYL_FWD RDSW
86    LD      X2B  ; Cyl_Rev_Reed    Switch
      OUT     M43  ; PLC CYL_REV RDSW
88    LD      X2C  ; PLC PANEL SPARE 07
      OUT     M44  ; PLC PANEL SPARE 07
90    LD      X2D  ; PLC PANEL SPARE 08
      OUT     M45  ; PLC PANEL SPARE 08
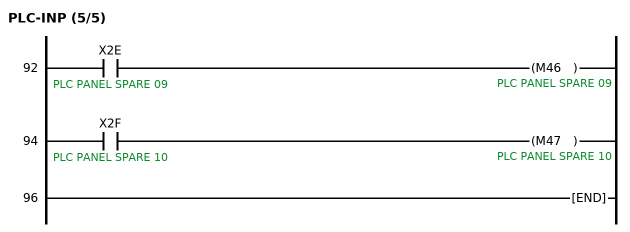
92    LD      X2E  ; PLC PANEL SPARE 09
      OUT     M46  ; PLC PANEL SPARE 09
94    LD      X2F  ; PLC PANEL SPARE 10
      OUT     M47  ; PLC PANEL SPARE 10
96    END
END_PROGRAM

// device comments not shown above
M251  ; RBT CYCLE START
M252  ; RSR
M253  ; WORK COMPLETE FROM RBT
M254  ; ROBOT HEALTHY IN RESUME
M255  ; PLC HEALTHY
M364  ; DO65
M365  ; DO66
M366  ; DO67
M367  ; DO68
M368  ; DO69
M369  ; DO70
M604  ; CYCLE START TO M/C
M605  ; M/C HEALTHY TO PLC
M606  ; STOPPER UP CMD TO M/C
M607  ; STOPPER DOWN CMD TO M/C
M608  ; JOB CLAMP CMD TO M/C
M609  ; JOB DECLAMP CMD TO M/C
M610  ; M/C READY FOR CYCLE START TO PLC
M650  ; M/C HEALTHY TO PLC
M651  ; M/C JOB COMPLETE TO PLC
M652  ; M/C JOB UNLOAD TO PLC
M653  ; READY TO DROP O/P PALLET
M654  ; READY TO PICK FROM M/C
M730  ; HMI PRODUCTION STOP
M900  ; HMI_EMG PRESSES _ALARM
M901  ; HMI_SAFETY DOOR EMG PRESSE_ALARM
M902  ; HMI_SAFETY DOOR OPEN_ALARM
M903  ; HMI_MACHINE FAULT_ALARM
M904  ; HMI_ROBOT FAULT _ALARM
M905  ; HMI_RBT DANGER ZONE_ALARM
